// Mitsubishi GX Works2 project: 동작   PLC: Q02/Q02H

PROGRAM MAIN
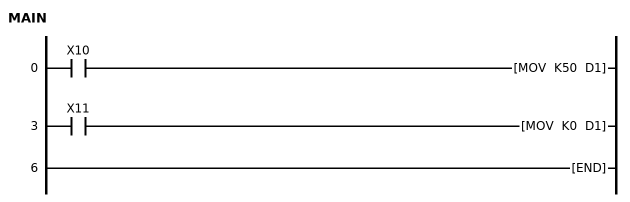
0     LD      X10
      MOV     K50 D1
3     LD      X11
      MOV     K0 D1
6     END
END_PROGRAM

PROGRAM MAIN1
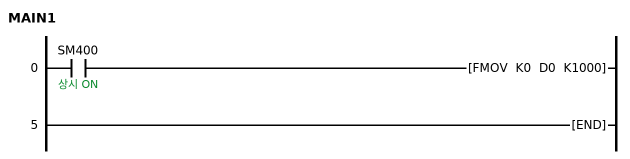
0     LD      SM400  ; 상시 ON
      FMOV    K0 D0 K1000
5     END
END_PROGRAM
